FUNCTION_BLOCK TeknicEIP_old_2
VAR_INPUT CONSTANT
	bEnable : BOOL;
END_VAR
VAR_OUTPUT
	enable AT %Q* : BOOL; //enable + pulses
	A AT %Q* : BOOL; //direction (F = inwards, T = outwards)
	B AT %Q* : BOOL; //home bit
	brakeRelease AT %Q* : BOOL;
	
	contact AT %I* : BOOL;
	
	home AT %I* : BOOL;
	outerLimit AT %I* : BOOL;
	innerLimit AT %I* : BOOL;
	done AT %I* : BOOL;	
	
	homeSet : BOOL;
	busy : BOOL;
	error : BOOL;
	
	position : REAL;
END_VAR
VAR
	mode : (IDLE, TARGET, CONTINUOUS);
	
	pulser : TON;	
	requestedPulses : INT;
	
	step : Homing;//(IDLE, HOME_UP, HOME_FINAL, DOWN, REDO_HOME, HOME_DONE);
END_VAR
VAR_STAT CONSTANT
	pulseWidth : TIME := T#25MS;
	unitsPerPulse : INT := 800; //800 Teknic units per revolution
	distancePerPulse : INT := 5; //5mm per revolution
END_VAR

enable := bEnable;
IF NOT bEnable THEN
	RETURN;
END_IF

pulser(IN:= , PT:= pulseWidth, Q=> , ET=> ); //when timer is enabled, this toggles enable every <pulseWidth>

IF requestedPulses = 0 THEN
	busy := FALSE;
	
	enable := TRUE;
	pulser.IN := FALSE;
	RETURN;
END_IF

busy := TRUE;
pulser.IN := TRUE;

IF pulser.Q THEN
	pulser.IN := FALSE;
	enable := NOT enable;
	
	IF enable THEN //enable is TRUE after toggle
		requestedPulses := requestedPulses - 1;
		
		IF A THEN
			position := position + distancePerPulse;
		ELSE
			position := position - distancePerPulse;
		END_IF
	END_IF
	
END_IF

(*
CASE mode OF
	IDLE:
		
	
	TARGET:
	

	CONTINUOUS:
		
		
		
END_CASE
*)

METHOD homingSequence : BOOL
CASE step OF
	Homing.IDLE:
		enable := FALSE;
		A := FALSE;
		B := FALSE;
		brakeRelease := TRUE;
		
		homeSet := FALSE;
		step := Homing.REDO;
		
	Homing.REDO: //let insertion drop to inner limit before homing
		enable := FALSE;
		A := FALSE;
		B := FALSE;
		brakeRelease := TRUE;
		
		IF NOT innerLimit THEN
			enable := TRUE;
			step := Homing.HOME_OUT;
		END_IF
	
	Homing.HOME_OUT:
		enable := TRUE;
		A := FALSE;
		B := TRUE;
		brakeRelease := TRUE;
		
		IF NOT home THEN
			B := FALSE;
			step := Homing.DONE;
		END_IF
		
	Homing.DONE:
		enable := TRUE;
		A := FALSE;
		B := FALSE;
		brakeRelease := TRUE;
		
		position := 0;
		homeSet := TRUE;
		homingSequence := TRUE;
		step := Homing.IDLE;
	
END_CASE
END_METHOD

METHOD moveAbsolute : BOOL
VAR_INPUT
	target : REAL;
END_VAR
END_METHOD

METHOD PRIVATE requestPulses : BOOL
VAR_INPUT
	request : INT;
END_VAR
IF (done OR requestedPulses = 0) AND request > 0 THEN
	requestedPulses := request;
	
	requestPulses := TRUE;
END_IF
END_METHOD

METHOD reset : BOOL
VAR_INPUT
END_VAR
END_METHOD

METHOD traverse : BOOL
VAR_INPUT
	direction : BOOL; //direction (F = inwards, T = outwards)
END_VAR
A := direction;
traverse := requestPulses(1);
END_METHOD

END_FUNCTION_BLOCK

(* stored: Version 1.1.0.1, ProductVersion 3.1.4024.11
   POU TeknicEIP_old_2: Id {668f31ab-c32e-4358-82c0-60575d137515}, SpecialFunc None
   Method homingSequence: Id {de17b18a-5b16-4271-bf39-f9d8af0e059d}
   Method moveAbsolute: Id {2330c12a-66d8-40f0-94c2-bdd4a06c20ee}
   Method requestPulses: Id {86f56a01-7fff-4f91-a0ab-1355c6f2262d}
   Method reset: Id {f33e4416-7cea-4ad8-9ff4-0e1a44f1ced7}
   Method traverse: Id {b8282b74-25fa-40ac-93c2-963bfe91f1d1} *)
